// TIA Portal V21 export
FUNCTION_BLOCK "FB310"   // FB310, LAD
TITLE = FB310
{ S7_Optimized_Access := 'TRUE' }
AUTHOR : PRECISE
FAMILY : PRECISE
// RAW MATERIAL ADDITION 
// 0-MANUAL/1-SUCTION/2-LIQUID DRUM
// stored: AutoNumber false, MemoryReserve 100, SetENOAutomatically false
   VAR_INPUT
      Enable : Bool;
      Disable : Bool;
      Fault : Bool;
      SecPulse : Bool;
      AlwaysTrue : Bool;
      StartConfirmationPopupSel : Bool;   // StartConfirmationPopupSel: 0-NO/1-YES
      EndConfirmationPopupSel : Bool;   // EndConfirmationPopupSel: 0-NO/1-YES
      RMAddTypeSel : Int;   // RMAddTypeSel: 0-Manual/1-Suction/2-Liquid Drum
      RMTypeSel : Int := 1;   // RM Type Sel: Graules or Flakes -0/FinePowder-1
      WeightBasedSel : Bool;   // Weight Based Sel: 0-NO/1-YES
      AdditionMethodSel : Bool;   // Addition Method : 0-Add In Weight/1-Loss In Weight
      RMAddPopupSel : Bool;   // RM Add Popup Sel: 0-NO/1-YES
      SetRMNo : Int := 1;
      "SetVacuum/SetPressure" : Real := -300.0;   // SetVauum - For unit "mmHg" / SetPressure - For unit "bar"
      SetQuantity : Real := 10.0;   // Weight Based Sel: 1-YES
      SetSpeed : Real := 50.0;
      "ActualVacuum/ActualPressure" : Real;   // ActualVauum - For unit "mmHg" / ActualPressure - For unit "bar"
      ActualQuantity : Real;   // Collecting Vessel Weight
      ActualQuantityRMVessel : Real;   // Transffering Vessel Weight
      "VacuumTol/PressureTol" : Real := 10.0;   // VacuumTol - For unit "mmHg" / PressureTol - For unit "bar"
      DelaytoSettleMaterial : Int := 5;
      InflightQuantitySuction : Real;
      InflightQuantityLiqDrum : Real;
      DelaytoStartPump : Int := 3;
   END_VAR
   VAR_OUTPUT
      VacuumInValve : Bool;
      VacuumLineValves : Bool;
      SuctionInValve : Bool;
      VacuumPumpCmd : Bool;
      LineValves : Bool;
      PumpCmd : Bool;
      StartConfirmationPopup : Bool;   // For Start Confirmation Popup Selection: Yes
      EndConfirmationPopup : Bool;   // For End Confirmation Popup Selection: Yes
      DelaytoSettleMaterialPopup : Bool;   // "WAITING FOR MATERIAL TO SETTLE"
      RMAddPopup : Bool;   // For RMAddPopupSel: 1-YES
      RMAddPopupManual : Bool;   // For RMAddPopupSel: 1-YES
      ActualSpeed : Real;
      VisibleRM1 : Bool;
      VisibleRM2 : Bool;
      VisibleRM3 : Bool;
      VisibleRM4 : Bool;
      VisibleRM5 : Bool;
      VisibleRM6 : Bool;
      VisibleRM7 : Bool;
      VisibleRM8 : Bool;
      VisibleRM9 : Bool;
      VisibleRM10 : Bool;
      PrintTrigger : Bool;
      PrintWord : Int;
      PrintStatus : String[50];
   END_VAR
   VAR_IN_OUT
      Start : Bool;
      Stop : Bool;
      Reset : Bool;
      StartConfirmationAck : Bool;   // For Start Confirmation Popup Selection: Yes
      EndConfirmationAck : Bool;   // For End Confirmation Popup Selection: Yes
      SpareBtn1 : Bool;
      SpareBtn2 : Bool;
      Running : Bool;
      Selected : Bool;
      Paused : Bool;
      StartConfirmationPopupTemp : Bool;   // For Start Confirmation Popup Selection: Yes
      EndConfirmationPopupTemp : Bool;   // For End Confirmation Popup Selection: Yes
      RMAddPopupTemp : Bool;   // For RMAddPopupSel: 1-YES
      RMAddStarted : Bool;
      RMAddOver : Bool;
      ActualSetQuantityCalc : Real;   // For WeightBaseSel: 1-YES
      ActualSetQuantity : Real;   // For WeightBaseSel: 1-YES
      RMAddAck1 : Bool;   // For RMAddPopupSel: 1-YES
      RMAddAck2 : Bool;   // For RMAddPopupSel: 1-YES
      RMAddAck3 : Bool;   // For RMAddPopupSel: 1-YES
      RMAddAck4 : Bool;   // For RMAddPopupSel: 1-YES
      RMAddAck5 : Bool;   // For RMAddPopupSel: 1-YES
      RMAddAck6 : Bool;   // For RMAddPopupSel: 1-YES
      RMAddAck7 : Bool;   // For RMAddPopupSel: 1-YES
      RMAddAck8 : Bool;   // For RMAddPopupSel: 1-YES
      RMAddAck9 : Bool;   // For RMAddPopupSel: 1-YES
      RMAddAck10 : Bool;   // For RMAddPopupSel: 1-YES
   END_VAR
   VAR
      PrintTriggerTemp : Bool;
      RE1 : Bool;
      RE2 : Bool;
      RE3 : Bool;
      RE4 : Bool;
      RE5 : Bool;
      RE6 : Bool;
      RE7 : Bool;
      RE8 : Bool;
      RE9 : Bool;
      RE10 : Bool;
      RE11 : Bool;
      PrintTriggerResetTimer { S7_SetPoint := 'True'} : TON_TIME;
      BtnResetTimer { S7_SetPoint := 'True'} : TON_TIME;
   END_VAR
   VAR RETAIN
      NameRM1 : String[100];
   END_VAR
   VAR
      NameRM2 : String[100];
      NameRM3 : String[100];
      NameRM4 : String[100];
      NameRM5 : String[100];
      NameRM6 : String[100];
      NameRM7 : String[100];
      NameRM8 : String[100];
      NameRM9 : String[100];
      NameRM10 : String[100];
      Manual { S7_SetPoint := 'True'} : "FB307";
      Suction { S7_SetPoint := 'True'} : "FB308";
      LiqDrum { S7_SetPoint := 'True'} : "FB309";
   END_VAR
   VAR_TEMP
      STATUS1 : String[40];
      STATUS2 : String[40];
      STATUS3 : String[40];
      STATUS4 : String[40];
      STATUS5 : String[40];
      Blank : String[40];
   END_VAR
   VAR_TEMP   // added for the SCL form of the ladder/FBD networks
      _w1 : Bool;
      _w2 : Bool;
      _w3 : Bool;
      _w4 : Bool;
      _w5 : Bool;
      _w6 : Bool;
   END_VAR
BEGIN

REGION Network 1: Running
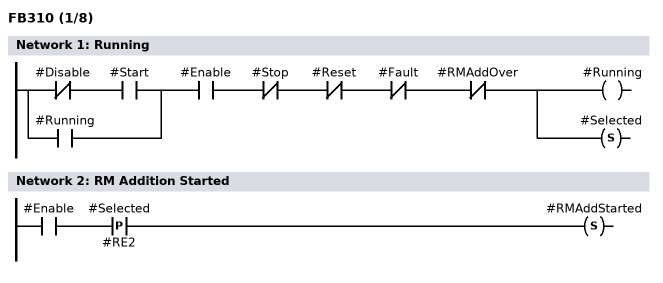
   RUNG wire#powerrail
      I_Contact( #Disable )
      Contact( #Start )
      wire#w1
      Contact( #Enable )
      I_Contact( #Stop )
      I_Contact( #Reset )
      I_Contact( #Fault )
      I_Contact( #RMAddOver )
      wire#w2
      Coil( #Running )
   END_RUNG
   RUNG wire#powerrail
      Contact( #Running )
   END_RUNG wire#w1
   RUNG wire#w2
      S_Coil( #Selected )
   END_RUNG
   // the same network as SCL:
   #Running := ((NOT #Disable AND #Start) OR #Running) AND #Enable AND NOT #Stop AND NOT #Reset AND NOT #Fault AND NOT #RMAddOver;
   IF #Running THEN #Selected := TRUE; END_IF;
END_REGION

REGION Network 2: RM Addition Started
   RUNG wire#powerrail
      Contact( #Enable )
      P_Contact(operand := #Selected, bit := #RE2)
      S_Coil( #RMAddStarted )
   END_RUNG
   // the same network as SCL:
   #_w1 := #Enable AND #Selected AND NOT #RE2;   // rising edge of #Selected
   #RE2 := #Selected;
   IF #_w1 THEN #RMAddStarted := TRUE; END_IF;
END_REGION

REGION Network 3: RM Addition Parameters
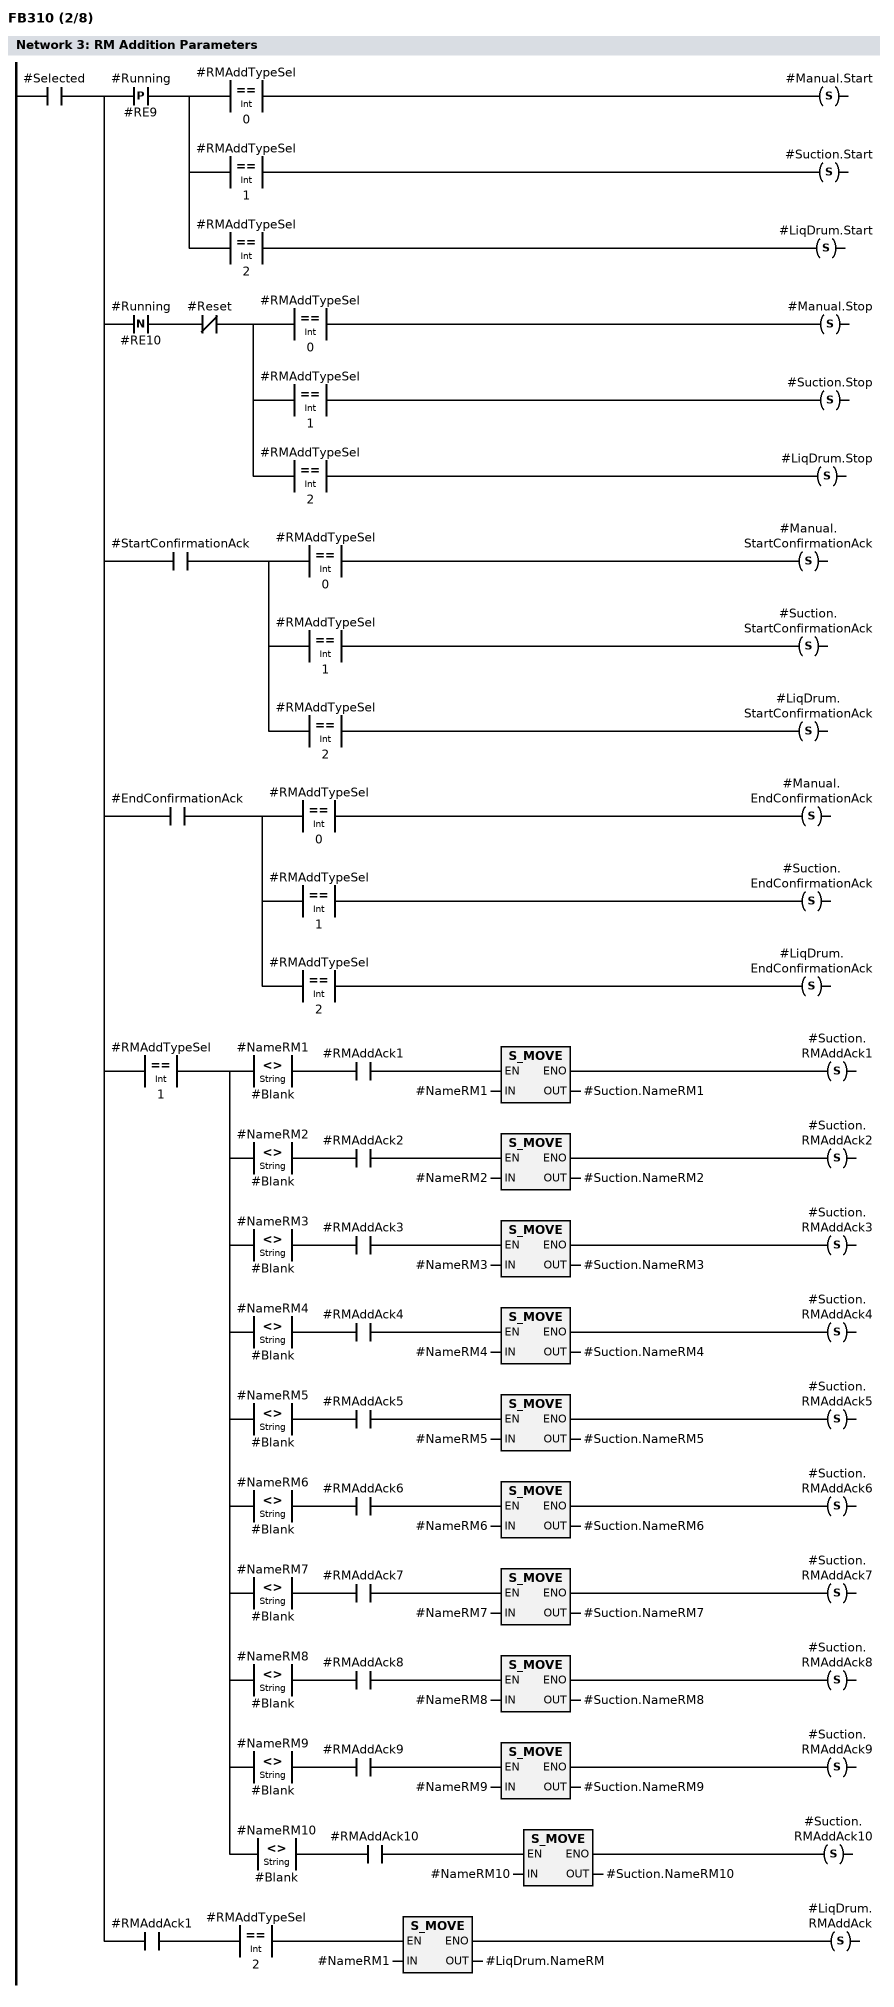
   RUNG wire#powerrail
      Contact( #Selected )
      wire#w1
      P_Contact(operand := #Running, bit := #RE9)
      wire#w2
      { S7_Templates := "SrcType := Int" } EQ_Contact(in1 := #RMAddTypeSel, in2 := 0)
      S_Coil( #Manual.Start )
   END_RUNG
   RUNG wire#w2
      { S7_Templates := "SrcType := Int" } EQ_Contact(in1 := #RMAddTypeSel, in2 := 1)
      S_Coil( #Suction.Start )
   END_RUNG
   RUNG wire#w2
      { S7_Templates := "SrcType := Int" } EQ_Contact(in1 := #RMAddTypeSel, in2 := 2)
      S_Coil( #LiqDrum.Start )
   END_RUNG
   RUNG wire#w1
      N_Contact(operand := #Running, bit := #RE10)
      I_Contact( #Reset )
      wire#w3
      { S7_Templates := "SrcType := Int" } EQ_Contact(in1 := #RMAddTypeSel, in2 := 0)
      S_Coil( #Manual.Stop )
   END_RUNG
   RUNG wire#w3
      { S7_Templates := "SrcType := Int" } EQ_Contact(in1 := #RMAddTypeSel, in2 := 1)
      S_Coil( #Suction.Stop )
   END_RUNG
   RUNG wire#w3
      { S7_Templates := "SrcType := Int" } EQ_Contact(in1 := #RMAddTypeSel, in2 := 2)
      S_Coil( #LiqDrum.Stop )
   END_RUNG
   RUNG wire#w1
      Contact( #StartConfirmationAck )
      wire#w4
      { S7_Templates := "SrcType := Int" } EQ_Contact(in1 := #RMAddTypeSel, in2 := 0)
      S_Coil( #Manual.StartConfirmationAck )
   END_RUNG
   RUNG wire#w4
      { S7_Templates := "SrcType := Int" } EQ_Contact(in1 := #RMAddTypeSel, in2 := 1)
      S_Coil( #Suction.StartConfirmationAck )
   END_RUNG
   RUNG wire#w4
      { S7_Templates := "SrcType := Int" } EQ_Contact(in1 := #RMAddTypeSel, in2 := 2)
      S_Coil( #LiqDrum.StartConfirmationAck )
   END_RUNG
   RUNG wire#w1
      Contact( #EndConfirmationAck )
      wire#w5
      { S7_Templates := "SrcType := Int" } EQ_Contact(in1 := #RMAddTypeSel, in2 := 0)
      S_Coil( #Manual.EndConfirmationAck )
   END_RUNG
   RUNG wire#w5
      { S7_Templates := "SrcType := Int" } EQ_Contact(in1 := #RMAddTypeSel, in2 := 1)
      S_Coil( #Suction.EndConfirmationAck )
   END_RUNG
   RUNG wire#w5
      { S7_Templates := "SrcType := Int" } EQ_Contact(in1 := #RMAddTypeSel, in2 := 2)
      S_Coil( #LiqDrum.EndConfirmationAck )
   END_RUNG
   RUNG wire#w1
      { S7_Templates := "SrcType := Int" } EQ_Contact(in1 := #RMAddTypeSel, in2 := 1)
      wire#w6
      { S7_Templates := "SrcType := String" } NE_Contact(in1 := #NameRM1, in2 := #Blank)
      Contact( #RMAddAck1 )
      S_Move(in := #NameRM1, out => #Suction.NameRM1)
      S_Coil( #Suction.RMAddAck1 )
   END_RUNG
   RUNG wire#w6
      { S7_Templates := "SrcType := String" } NE_Contact(in1 := #NameRM2, in2 := #Blank)
      Contact( #RMAddAck2 )
      S_Move(in := #NameRM2, out => #Suction.NameRM2)
      S_Coil( #Suction.RMAddAck2 )
   END_RUNG
   RUNG wire#w6
      { S7_Templates := "SrcType := String" } NE_Contact(in1 := #NameRM3, in2 := #Blank)
      Contact( #RMAddAck3 )
      S_Move(in := #NameRM3, out => #Suction.NameRM3)
      S_Coil( #Suction.RMAddAck3 )
   END_RUNG
   RUNG wire#w6
      { S7_Templates := "SrcType := String" } NE_Contact(in1 := #NameRM4, in2 := #Blank)
      Contact( #RMAddAck4 )
      S_Move(in := #NameRM4, out => #Suction.NameRM4)
      S_Coil( #Suction.RMAddAck4 )
   END_RUNG
   RUNG wire#w6
      { S7_Templates := "SrcType := String" } NE_Contact(in1 := #NameRM5, in2 := #Blank)
      Contact( #RMAddAck5 )
      S_Move(in := #NameRM5, out => #Suction.NameRM5)
      S_Coil( #Suction.RMAddAck5 )
   END_RUNG
   RUNG wire#w6
      { S7_Templates := "SrcType := String" } NE_Contact(in1 := #NameRM6, in2 := #Blank)
      Contact( #RMAddAck6 )
      S_Move(in := #NameRM6, out => #Suction.NameRM6)
      S_Coil( #Suction.RMAddAck6 )
   END_RUNG
   RUNG wire#w6
      { S7_Templates := "SrcType := String" } NE_Contact(in1 := #NameRM7, in2 := #Blank)
      Contact( #RMAddAck7 )
      S_Move(in := #NameRM7, out => #Suction.NameRM7)
      S_Coil( #Suction.RMAddAck7 )
   END_RUNG
   RUNG wire#w6
      { S7_Templates := "SrcType := String" } NE_Contact(in1 := #NameRM8, in2 := #Blank)
      Contact( #RMAddAck8 )
      S_Move(in := #NameRM8, out => #Suction.NameRM8)
      S_Coil( #Suction.RMAddAck8 )
   END_RUNG
   RUNG wire#w6
      { S7_Templates := "SrcType := String" } NE_Contact(in1 := #NameRM9, in2 := #Blank)
      Contact( #RMAddAck9 )
      S_Move(in := #NameRM9, out => #Suction.NameRM9)
      S_Coil( #Suction.RMAddAck9 )
   END_RUNG
   RUNG wire#w6
      { S7_Templates := "SrcType := String" } NE_Contact(in1 := #NameRM10, in2 := #Blank)
      Contact( #RMAddAck10 )
      S_Move(in := #NameRM10, out => #Suction.NameRM10)
      S_Coil( #Suction.RMAddAck10 )
   END_RUNG
   RUNG wire#w1
      Contact( #RMAddAck1 )
      { S7_Templates := "SrcType := Int" } EQ_Contact(in1 := #RMAddTypeSel, in2 := 2)
      S_Move(in := #NameRM1, out => #LiqDrum.NameRM)
      S_Coil( #LiqDrum.RMAddAck )
   END_RUNG
   // the same network as SCL:
   #_w1 := #Selected AND #Running AND NOT #RE9;   // rising edge of #Running
   #RE9 := #Running;
   IF #_w1 AND (#RMAddTypeSel = 0) THEN #Manual.Start := TRUE; END_IF;
   IF #_w1 AND (#RMAddTypeSel = 1) THEN #Suction.Start := TRUE; END_IF;
   IF #_w1 AND (#RMAddTypeSel = 2) THEN #LiqDrum.Start := TRUE; END_IF;
   #_w2 := #Selected AND NOT #Running AND #RE10;   // falling edge of #Running
   #RE10 := #Running;
   #_w3 := #_w2 AND NOT #Reset;
   IF #_w3 AND (#RMAddTypeSel = 0) THEN #Manual.Stop := TRUE; END_IF;
   IF #_w3 AND (#RMAddTypeSel = 1) THEN #Suction.Stop := TRUE; END_IF;
   IF #_w3 AND (#RMAddTypeSel = 2) THEN #LiqDrum.Stop := TRUE; END_IF;
   #_w4 := #Selected AND #StartConfirmationAck;
   IF #_w4 AND (#RMAddTypeSel = 0) THEN #Manual.StartConfirmationAck := TRUE; END_IF;
   IF #_w4 AND (#RMAddTypeSel = 1) THEN #Suction.StartConfirmationAck := TRUE; END_IF;
   IF #_w4 AND (#RMAddTypeSel = 2) THEN #LiqDrum.StartConfirmationAck := TRUE; END_IF;
   #_w5 := #Selected AND #EndConfirmationAck;
   IF #_w5 AND (#RMAddTypeSel = 0) THEN #Manual.EndConfirmationAck := TRUE; END_IF;
   IF #_w5 AND (#RMAddTypeSel = 1) THEN #Suction.EndConfirmationAck := TRUE; END_IF;
   IF #_w5 AND (#RMAddTypeSel = 2) THEN #LiqDrum.EndConfirmationAck := TRUE; END_IF;
   #_w6 := #Selected AND (#RMAddTypeSel = 1);
   IF #_w6 AND (#NameRM1 <> #Blank) AND #RMAddAck1 THEN
       #Suction.NameRM1 := #NameRM1;
       #Suction.RMAddAck1 := TRUE;
   END_IF;
   IF #_w6 AND (#NameRM2 <> #Blank) AND #RMAddAck2 THEN
       #Suction.NameRM2 := #NameRM2;
       #Suction.RMAddAck2 := TRUE;
   END_IF;
   IF #_w6 AND (#NameRM3 <> #Blank) AND #RMAddAck3 THEN
       #Suction.NameRM3 := #NameRM3;
       #Suction.RMAddAck3 := TRUE;
   END_IF;
   IF #_w6 AND (#NameRM4 <> #Blank) AND #RMAddAck4 THEN
       #Suction.NameRM4 := #NameRM4;
       #Suction.RMAddAck4 := TRUE;
   END_IF;
   IF #_w6 AND (#NameRM5 <> #Blank) AND #RMAddAck5 THEN
       #Suction.NameRM5 := #NameRM5;
       #Suction.RMAddAck5 := TRUE;
   END_IF;
   IF #_w6 AND (#NameRM6 <> #Blank) AND #RMAddAck6 THEN
       #Suction.NameRM6 := #NameRM6;
       #Suction.RMAddAck6 := TRUE;
   END_IF;
   IF #_w6 AND (#NameRM7 <> #Blank) AND #RMAddAck7 THEN
       #Suction.NameRM7 := #NameRM7;
       #Suction.RMAddAck7 := TRUE;
   END_IF;
   IF #_w6 AND (#NameRM8 <> #Blank) AND #RMAddAck8 THEN
       #Suction.NameRM8 := #NameRM8;
       #Suction.RMAddAck8 := TRUE;
   END_IF;
   IF #_w6 AND (#NameRM9 <> #Blank) AND #RMAddAck9 THEN
       #Suction.NameRM9 := #NameRM9;
       #Suction.RMAddAck9 := TRUE;
   END_IF;
   IF #_w6 AND (#NameRM10 <> #Blank) AND #RMAddAck10 THEN
       #Suction.NameRM10 := #NameRM10;
       #Suction.RMAddAck10 := TRUE;
   END_IF;
   IF #Selected AND #RMAddAck1 AND (#RMAddTypeSel = 2) THEN
       #LiqDrum.NameRM := #NameRM1;
       #LiqDrum.RMAddAck := TRUE;
   END_IF;
END_REGION

REGION Network 4: RM Addition Manual
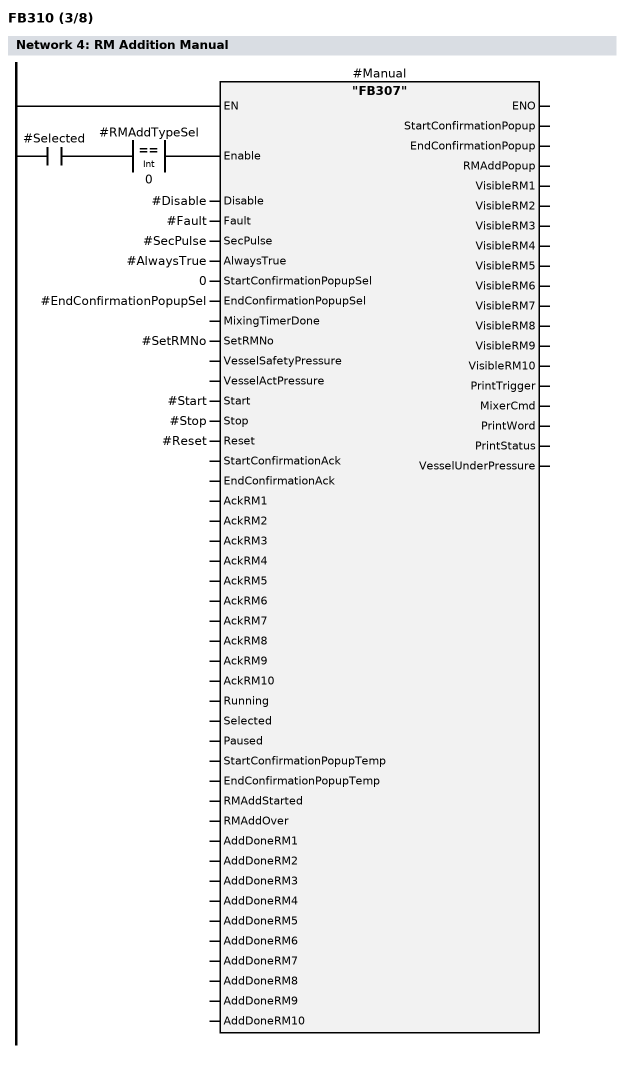
   RUNG wire#powerrail
      #Manual(Enable := wire#w1, Disable := #Disable, Fault := #Fault, SecPulse := #SecPulse, AlwaysTrue := #AlwaysTrue, StartConfirmationPopupSel := 0, EndConfirmationPopupSel := #EndConfirmationPopupSel, MixingTimerDone :=, SetRMNo := #SetRMNo, VesselSafetyPressure :=, VesselActPressure :=, Start := #Start, Stop := #Stop, Reset := #Reset, StartConfirmationAck :=, EndConfirmationAck :=, AckRM1 :=, AckRM2 :=, AckRM3 :=, AckRM4 :=, AckRM5 :=, AckRM6 :=, AckRM7 :=, AckRM8 :=, AckRM9 :=, AckRM10 :=, Running :=, Selected :=, Paused :=, StartConfirmationPopupTemp :=, EndConfirmationPopupTemp :=, RMAddStarted :=, RMAddOver :=, AddDoneRM1 :=, AddDoneRM2 :=, AddDoneRM3 :=, AddDoneRM4 :=, AddDoneRM5 :=, AddDoneRM6 :=, AddDoneRM7 :=, AddDoneRM8 :=, AddDoneRM9 :=, AddDoneRM10 :=, StartConfirmationPopup =>, EndConfirmationPopup =>, RMAddPopup =>, VisibleRM1 =>, VisibleRM2 =>, VisibleRM3 =>, VisibleRM4 =>, VisibleRM5 =>, VisibleRM6 =>, VisibleRM7 =>, VisibleRM8 =>, VisibleRM9 =>, VisibleRM10 =>, PrintTrigger =>, MixerCmd =>, PrintWord =>, PrintStatus =>, VesselUnderPressure =>)
   END_RUNG
   RUNG wire#powerrail
      Contact( #Selected )
      { S7_Templates := "SrcType := Int" } EQ_Contact(in1 := #RMAddTypeSel, in2 := 0)
   END_RUNG wire#w1
   // the same network as SCL:
   #Manual(Enable := #Selected AND (#RMAddTypeSel = 0),   // "FB307"
           Disable := #Disable,
           Fault := #Fault,
           SecPulse := #SecPulse,
           AlwaysTrue := #AlwaysTrue,
           StartConfirmationPopupSel := 0,
           EndConfirmationPopupSel := #EndConfirmationPopupSel,
           SetRMNo := #SetRMNo,
           Start := #Start,
           Stop := #Stop,
           Reset := #Reset);
END_REGION

REGION Network 5: RM Addition Suction
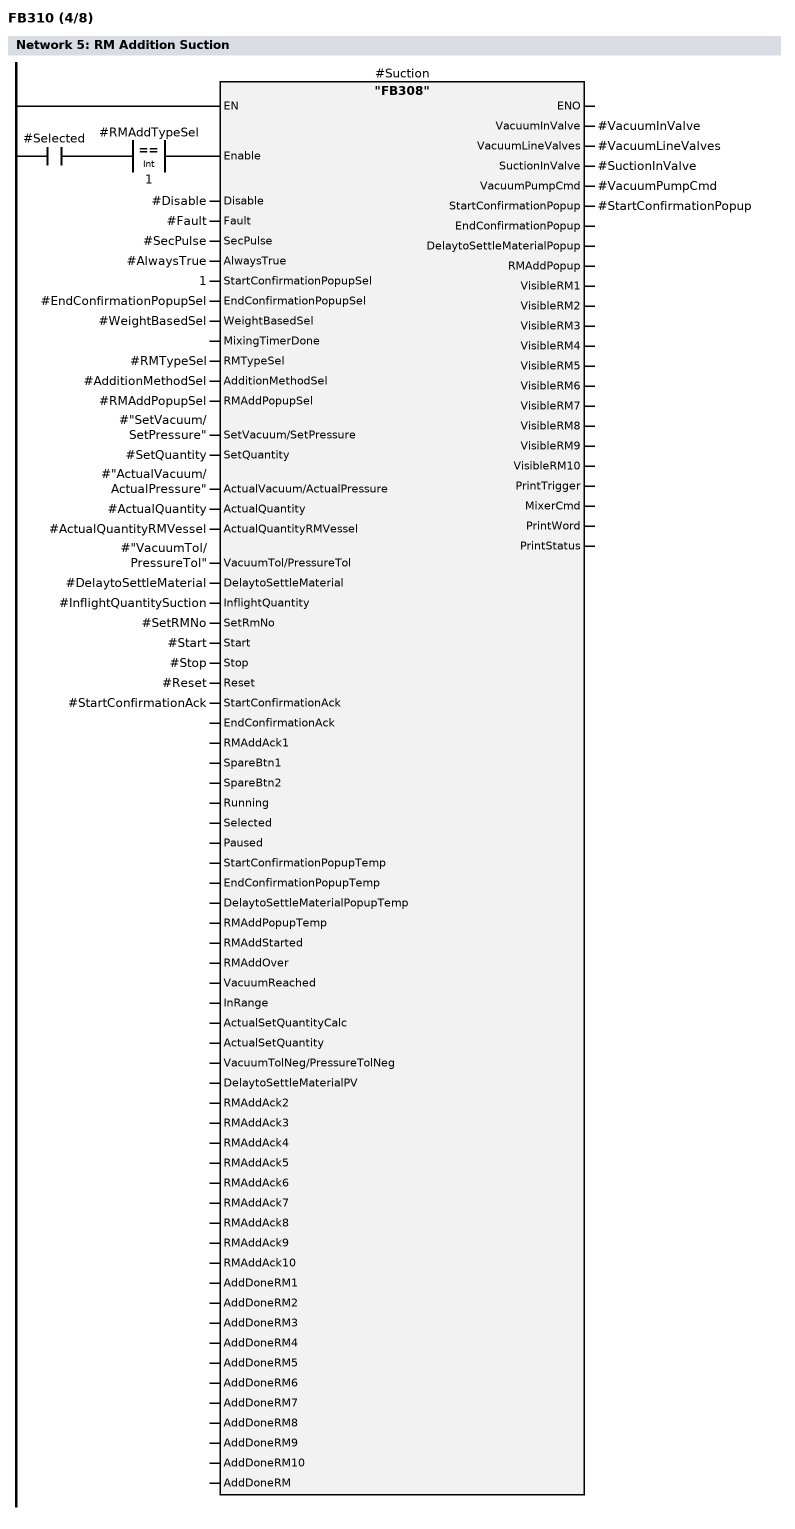
   RUNG wire#powerrail
      #Suction(Enable := wire#w1, Disable := #Disable, Fault := #Fault, SecPulse := #SecPulse, AlwaysTrue := #AlwaysTrue, StartConfirmationPopupSel := 1, EndConfirmationPopupSel := #EndConfirmationPopupSel, WeightBasedSel := #WeightBasedSel, MixingTimerDone :=, RMTypeSel := #RMTypeSel, AdditionMethodSel := #AdditionMethodSel, RMAddPopupSel := #RMAddPopupSel, "SetVacuum/SetPressure" := #"SetVacuum/SetPressure", SetQuantity := #SetQuantity, "ActualVacuum/ActualPressure" := #"ActualVacuum/ActualPressure", ActualQuantity := #ActualQuantity, ActualQuantityRMVessel := #ActualQuantityRMVessel, "VacuumTol/PressureTol" := #"VacuumTol/PressureTol", DelaytoSettleMaterial := #DelaytoSettleMaterial, InflightQuantity := #InflightQuantitySuction, SetRmNo := #SetRMNo, Start := #Start, Stop := #Stop, Reset := #Reset, StartConfirmationAck := #StartConfirmationAck, EndConfirmationAck :=, RMAddAck1 :=, SpareBtn1 :=, SpareBtn2 :=, Running :=, Selected :=, Paused :=, StartConfirmationPopupTemp :=, EndConfirmationPopupTemp :=, DelaytoSettleMaterialPopupTemp :=, RMAddPopupTemp :=, RMAddStarted :=, RMAddOver :=, VacuumReached :=, InRange :=, ActualSetQuantityCalc :=, ActualSetQuantity :=, "VacuumTolNeg/PressureTolNeg" :=, DelaytoSettleMaterialPV :=, RMAddAck2 :=, RMAddAck3 :=, RMAddAck4 :=, RMAddAck5 :=, RMAddAck6 :=, RMAddAck7 :=, RMAddAck8 :=, RMAddAck9 :=, RMAddAck10 :=, AddDoneRM1 :=, AddDoneRM2 :=, AddDoneRM3 :=, AddDoneRM4 :=, AddDoneRM5 :=, AddDoneRM6 :=, AddDoneRM7 :=, AddDoneRM8 :=, AddDoneRM9 :=, AddDoneRM10 :=, AddDoneRM :=, VacuumInValve => #VacuumInValve, VacuumLineValves => #VacuumLineValves, SuctionInValve => #SuctionInValve, VacuumPumpCmd => #VacuumPumpCmd, StartConfirmationPopup => #StartConfirmationPopup, EndConfirmationPopup =>, DelaytoSettleMaterialPopup =>, RMAddPopup =>, VisibleRM1 =>, VisibleRM2 =>, VisibleRM3 =>, VisibleRM4 =>, VisibleRM5 =>, VisibleRM6 =>, VisibleRM7 =>, VisibleRM8 =>, VisibleRM9 =>, VisibleRM10 =>, PrintTrigger =>, MixerCmd =>, PrintWord =>, PrintStatus =>)
   END_RUNG
   RUNG wire#powerrail
      Contact( #Selected )
      { S7_Templates := "SrcType := Int" } EQ_Contact(in1 := #RMAddTypeSel, in2 := 1)
   END_RUNG wire#w1
   // the same network as SCL:
   #Suction(Enable := #Selected AND (#RMAddTypeSel = 1),   // "FB308"
            Disable := #Disable,
            Fault := #Fault,
            SecPulse := #SecPulse,
            AlwaysTrue := #AlwaysTrue,
            StartConfirmationPopupSel := 1,
            EndConfirmationPopupSel := #EndConfirmationPopupSel,
            WeightBasedSel := #WeightBasedSel,
            RMTypeSel := #RMTypeSel,
            AdditionMethodSel := #AdditionMethodSel,
            RMAddPopupSel := #RMAddPopupSel,
            "SetVacuum/SetPressure" := #"SetVacuum/SetPressure",
            SetQuantity := #SetQuantity,
            "ActualVacuum/ActualPressure" := #"ActualVacuum/ActualPressure",
            ActualQuantity := #ActualQuantity,
            ActualQuantityRMVessel := #ActualQuantityRMVessel,
            "VacuumTol/PressureTol" := #"VacuumTol/PressureTol",
            DelaytoSettleMaterial := #DelaytoSettleMaterial,
            InflightQuantity := #InflightQuantitySuction,
            SetRmNo := #SetRMNo,
            Start := #Start,
            Stop := #Stop,
            Reset := #Reset,
            StartConfirmationAck := #StartConfirmationAck,
            VacuumInValve => #VacuumInValve,
            VacuumLineValves => #VacuumLineValves,
            SuctionInValve => #SuctionInValve,
            VacuumPumpCmd => #VacuumPumpCmd,
            StartConfirmationPopup => #StartConfirmationPopup);
END_REGION

REGION Network 6: RM Addition Liquid Drum
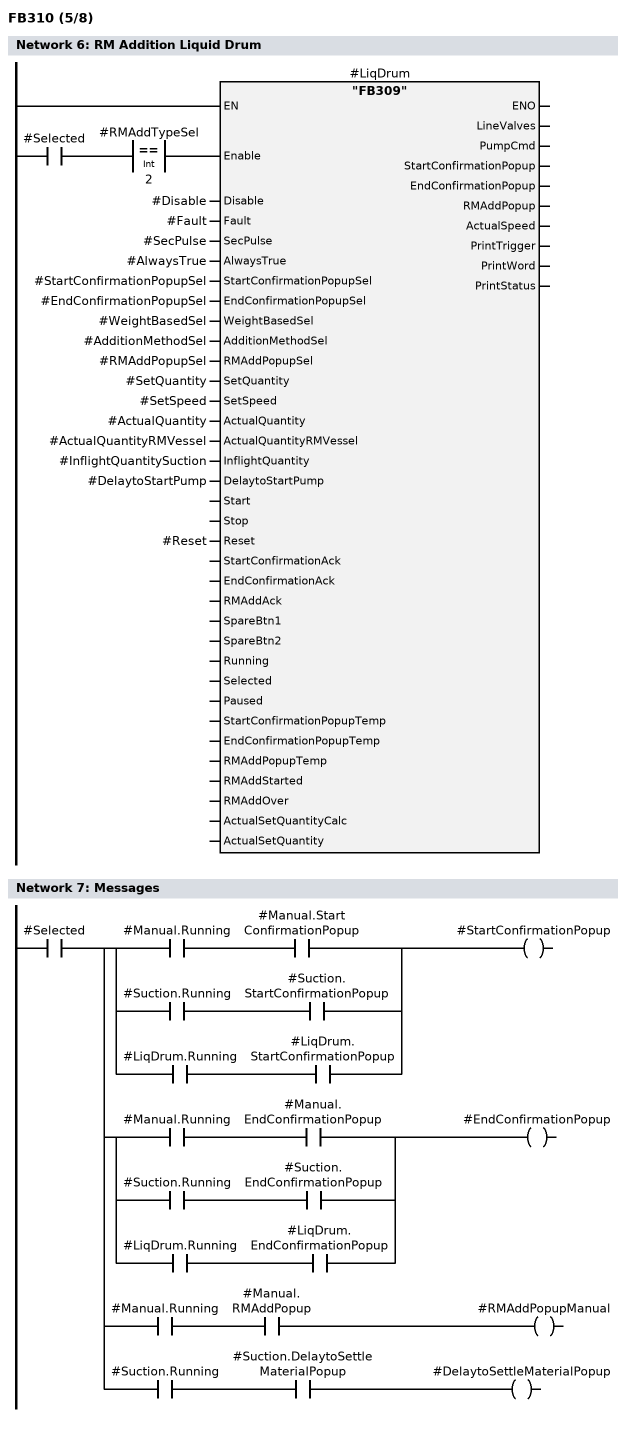
   RUNG wire#powerrail
      #LiqDrum(Enable := wire#w1, Disable := #Disable, Fault := #Fault, SecPulse := #SecPulse, AlwaysTrue := #AlwaysTrue, StartConfirmationPopupSel := #StartConfirmationPopupSel, EndConfirmationPopupSel := #EndConfirmationPopupSel, WeightBasedSel := #WeightBasedSel, AdditionMethodSel := #AdditionMethodSel, RMAddPopupSel := #RMAddPopupSel, SetQuantity := #SetQuantity, SetSpeed := #SetSpeed, ActualQuantity := #ActualQuantity, ActualQuantityRMVessel := #ActualQuantityRMVessel, InflightQuantity := #InflightQuantitySuction, DelaytoStartPump := #DelaytoStartPump, Start :=, Stop :=, Reset := #Reset, StartConfirmationAck :=, EndConfirmationAck :=, RMAddAck :=, SpareBtn1 :=, SpareBtn2 :=, Running :=, Selected :=, Paused :=, StartConfirmationPopupTemp :=, EndConfirmationPopupTemp :=, RMAddPopupTemp :=, RMAddStarted :=, RMAddOver :=, ActualSetQuantityCalc :=, ActualSetQuantity :=, LineValves =>, PumpCmd =>, StartConfirmationPopup =>, EndConfirmationPopup =>, RMAddPopup =>, ActualSpeed =>, PrintTrigger =>, PrintWord =>, PrintStatus =>)
   END_RUNG
   RUNG wire#powerrail
      Contact( #Selected )
      { S7_Templates := "SrcType := Int" } EQ_Contact(in1 := #RMAddTypeSel, in2 := 2)
   END_RUNG wire#w1
   // the same network as SCL:
   #LiqDrum(Enable := #Selected AND (#RMAddTypeSel = 2),   // "FB309"
            Disable := #Disable,
            Fault := #Fault,
            SecPulse := #SecPulse,
            AlwaysTrue := #AlwaysTrue,
            StartConfirmationPopupSel := #StartConfirmationPopupSel,
            EndConfirmationPopupSel := #EndConfirmationPopupSel,
            WeightBasedSel := #WeightBasedSel,
            AdditionMethodSel := #AdditionMethodSel,
            RMAddPopupSel := #RMAddPopupSel,
            SetQuantity := #SetQuantity,
            SetSpeed := #SetSpeed,
            ActualQuantity := #ActualQuantity,
            ActualQuantityRMVessel := #ActualQuantityRMVessel,
            InflightQuantity := #InflightQuantitySuction,
            DelaytoStartPump := #DelaytoStartPump,
            Reset := #Reset);
END_REGION

REGION Network 7: Messages
   RUNG wire#powerrail
      Contact( #Selected )
      wire#w1
      Contact( #Manual.Running )
      Contact( #Manual.StartConfirmationPopup )
      wire#w2
      Coil( #StartConfirmationPopup )
   END_RUNG
   RUNG wire#w1
      Contact( #Suction.Running )
      Contact( #Suction.StartConfirmationPopup )
   END_RUNG wire#w2
   RUNG wire#w1
      Contact( #LiqDrum.Running )
      Contact( #LiqDrum.StartConfirmationPopup )
   END_RUNG wire#w2
   RUNG wire#w1
      Contact( #Manual.Running )
      Contact( #Manual.EndConfirmationPopup )
      wire#w3
      Coil( #EndConfirmationPopup )
   END_RUNG
   RUNG wire#w1
      Contact( #Suction.Running )
      Contact( #Suction.EndConfirmationPopup )
   END_RUNG wire#w3
   RUNG wire#w1
      Contact( #LiqDrum.Running )
      Contact( #LiqDrum.EndConfirmationPopup )
   END_RUNG wire#w3
   RUNG wire#w1
      Contact( #Manual.Running )
      Contact( #Manual.RMAddPopup )
      Coil( #RMAddPopupManual )
   END_RUNG
   RUNG wire#w1
      Contact( #Suction.Running )
      Contact( #Suction.DelaytoSettleMaterialPopup )
      Coil( #DelaytoSettleMaterialPopup )
   END_RUNG
   // the same network as SCL:
   #StartConfirmationPopup := #Selected AND ((#Manual.Running AND #Manual.StartConfirmationPopup) OR (#Suction.Running AND #Suction.StartConfirmationPopup) OR (#LiqDrum.Running AND #LiqDrum.StartConfirmationPopup));
   #EndConfirmationPopup := #Selected AND ((#Manual.Running AND #Manual.EndConfirmationPopup) OR (#Suction.Running AND #Suction.EndConfirmationPopup) OR (#LiqDrum.Running AND #LiqDrum.EndConfirmationPopup));
   #RMAddPopupManual := #Selected AND #Manual.Running AND #Manual.RMAddPopup;
   #DelaytoSettleMaterialPopup := #Selected AND #Suction.Running AND #Suction.DelaytoSettleMaterialPopup;
END_REGION

REGION Network 8: Output
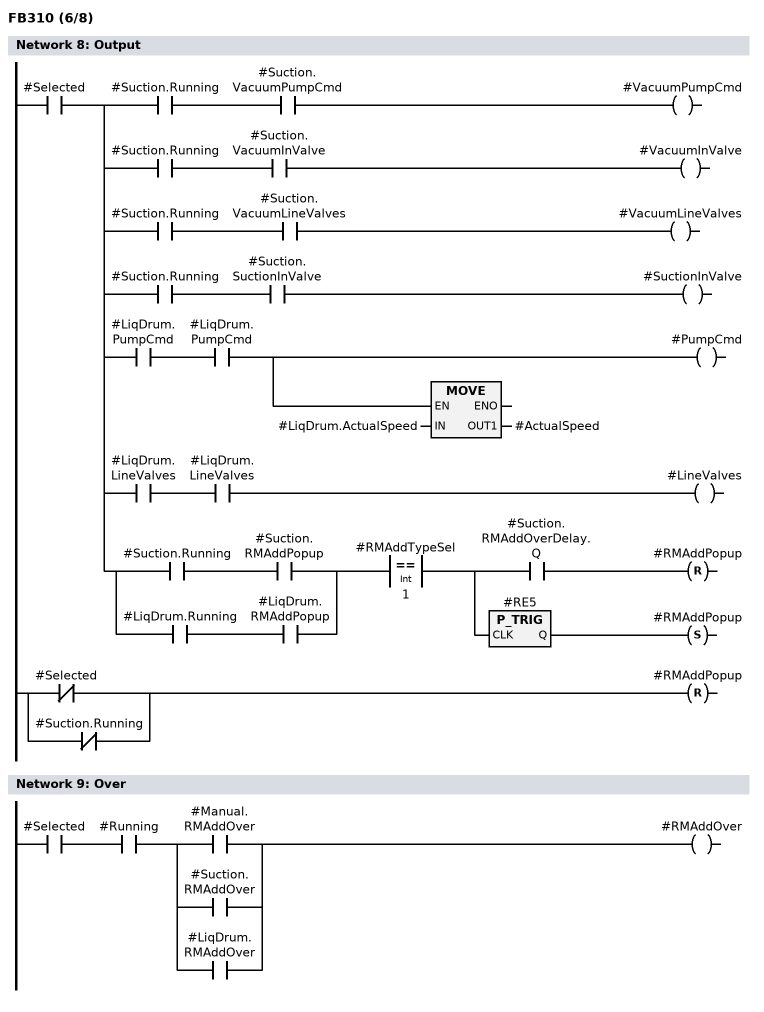
   RUNG wire#powerrail
      Contact( #Selected )
      wire#w1
      Contact( #Suction.Running )
      Contact( #Suction.VacuumPumpCmd )
      Coil( #VacuumPumpCmd )
   END_RUNG
   RUNG wire#w1
      Contact( #Suction.Running )
      Contact( #Suction.VacuumInValve )
      Coil( #VacuumInValve )
   END_RUNG
   RUNG wire#w1
      Contact( #Suction.Running )
      Contact( #Suction.VacuumLineValves )
      Coil( #VacuumLineValves )
   END_RUNG
   RUNG wire#w1
      Contact( #Suction.Running )
      Contact( #Suction.SuctionInValve )
      Coil( #SuctionInValve )
   END_RUNG
   RUNG wire#w1
      Contact( #LiqDrum.PumpCmd )
      Contact( #LiqDrum.PumpCmd )
      wire#w2
      Coil( #PumpCmd )
   END_RUNG
   RUNG wire#w2
      Move(in := #LiqDrum.ActualSpeed, out1 => #ActualSpeed)
   END_RUNG
   RUNG wire#w1
      Contact( #LiqDrum.LineValves )
      Contact( #LiqDrum.LineValves )
      Coil( #LineValves )
   END_RUNG
   RUNG wire#w1
      Contact( #Suction.Running )
      Contact( #Suction.RMAddPopup )
      wire#w3
      { S7_Templates := "SrcType := Int" } EQ_Contact(in1 := #RMAddTypeSel, in2 := 1)
      wire#w4
      Contact( #Suction.RMAddOverDelay.Q )
      R_Coil( #RMAddPopup )
   END_RUNG
   RUNG wire#w1
      Contact( #LiqDrum.Running )
      Contact( #LiqDrum.RMAddPopup )
   END_RUNG wire#w3
   RUNG wire#w4
      P_Trig( #RE5 )
      S_Coil( #RMAddPopup )
   END_RUNG
   RUNG wire#powerrail
      I_Contact( #Selected )
      wire#w5
      R_Coil( #RMAddPopup )
   END_RUNG
   RUNG wire#powerrail
      I_Contact( #Suction.Running )
   END_RUNG wire#w5
   // the same network as SCL:
   #VacuumPumpCmd := #Selected AND #Suction.Running AND #Suction.VacuumPumpCmd;
   #VacuumInValve := #Selected AND #Suction.Running AND #Suction.VacuumInValve;
   #VacuumLineValves := #Selected AND #Suction.Running AND #Suction.VacuumLineValves;
   #SuctionInValve := #Selected AND #Suction.Running AND #Suction.SuctionInValve;
   #PumpCmd := #Selected AND #LiqDrum.PumpCmd AND #LiqDrum.PumpCmd;
   IF #PumpCmd THEN #ActualSpeed := #LiqDrum.ActualSpeed; END_IF;
   #LineValves := #Selected AND #LiqDrum.LineValves AND #LiqDrum.LineValves;
   #_w1 := #Selected AND ((#Suction.Running AND #Suction.RMAddPopup) OR (#LiqDrum.Running AND #LiqDrum.RMAddPopup)) AND (#RMAddTypeSel = 1);
   IF #_w1 AND #Suction.RMAddOverDelay.Q THEN #RMAddPopup := FALSE; END_IF;
   #_w2 := #_w1 AND NOT #RE5;   // rising edge
   #RE5 := #_w1;
   IF #_w2 THEN #RMAddPopup := TRUE; END_IF;
   IF NOT #Selected OR NOT #Suction.Running THEN #RMAddPopup := FALSE; END_IF;
END_REGION

REGION Network 9: Over
   RUNG wire#powerrail
      Contact( #Selected )
      Contact( #Running )
      wire#w1
      Contact( #Manual.RMAddOver )
      wire#w2
      Coil( #RMAddOver )
   END_RUNG
   RUNG wire#w1
      Contact( #Suction.RMAddOver )
   END_RUNG wire#w2
   RUNG wire#w1
      Contact( #LiqDrum.RMAddOver )
   END_RUNG wire#w2
   // the same network as SCL:
   #RMAddOver := #Selected AND #Running AND (#Manual.RMAddOver OR #Suction.RMAddOver OR #LiqDrum.RMAddOver);
END_REGION

REGION Network 10: Print Status
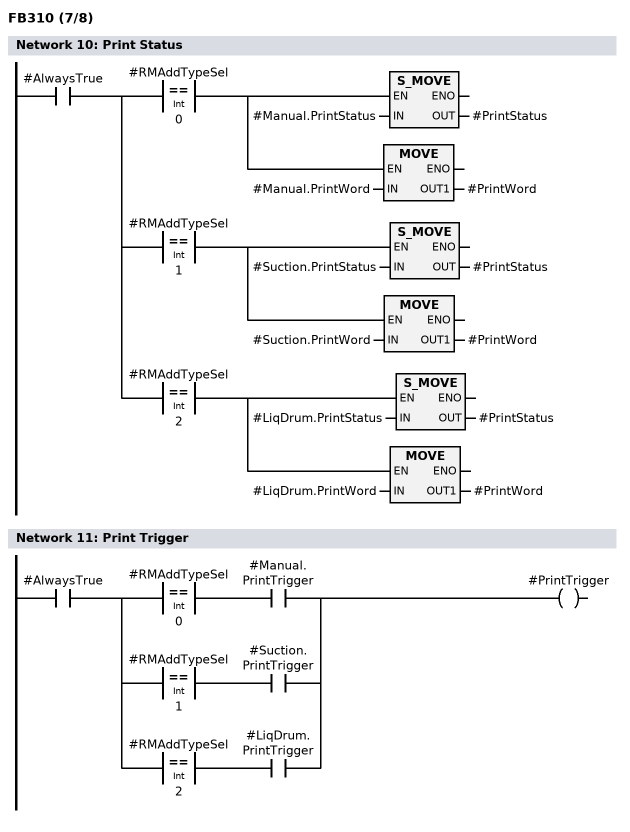
   RUNG wire#powerrail
      Contact( #AlwaysTrue )
      wire#w1
      { S7_Templates := "SrcType := Int" } EQ_Contact(in1 := #RMAddTypeSel, in2 := 0)
      wire#w2
      S_Move(in := #Manual.PrintStatus, out => #PrintStatus)
   END_RUNG
   RUNG wire#w2
      Move(in := #Manual.PrintWord, out1 => #PrintWord)
   END_RUNG
   RUNG wire#w1
      { S7_Templates := "SrcType := Int" } EQ_Contact(in1 := #RMAddTypeSel, in2 := 1)
      wire#w3
      S_Move(in := #Suction.PrintStatus, out => #PrintStatus)
   END_RUNG
   RUNG wire#w3
      Move(in := #Suction.PrintWord, out1 => #PrintWord)
   END_RUNG
   RUNG wire#w1
      { S7_Templates := "SrcType := Int" } EQ_Contact(in1 := #RMAddTypeSel, in2 := 2)
      wire#w4
      S_Move(in := #LiqDrum.PrintStatus, out => #PrintStatus)
   END_RUNG
   RUNG wire#w4
      Move(in := #LiqDrum.PrintWord, out1 => #PrintWord)
   END_RUNG
   // the same network as SCL:
   IF #AlwaysTrue AND (#RMAddTypeSel = 0) THEN
       #PrintStatus := #Manual.PrintStatus;
       #PrintWord := #Manual.PrintWord;
   END_IF;
   IF #AlwaysTrue AND (#RMAddTypeSel = 1) THEN
       #PrintStatus := #Suction.PrintStatus;
       #PrintWord := #Suction.PrintWord;
   END_IF;
   IF #AlwaysTrue AND (#RMAddTypeSel = 2) THEN
       #PrintStatus := #LiqDrum.PrintStatus;
       #PrintWord := #LiqDrum.PrintWord;
   END_IF;
END_REGION

REGION Network 11: Print Trigger
   RUNG wire#powerrail
      Contact( #AlwaysTrue )
      wire#w1
      { S7_Templates := "SrcType := Int" } EQ_Contact(in1 := #RMAddTypeSel, in2 := 0)
      Contact( #Manual.PrintTrigger )
      wire#w2
      Coil( #PrintTrigger )
   END_RUNG
   RUNG wire#w1
      { S7_Templates := "SrcType := Int" } EQ_Contact(in1 := #RMAddTypeSel, in2 := 1)
      Contact( #Suction.PrintTrigger )
   END_RUNG wire#w2
   RUNG wire#w1
      { S7_Templates := "SrcType := Int" } EQ_Contact(in1 := #RMAddTypeSel, in2 := 2)
      Contact( #LiqDrum.PrintTrigger )
   END_RUNG wire#w2
   // the same network as SCL:
   #PrintTrigger := #AlwaysTrue AND (((#RMAddTypeSel = 0) AND #Manual.PrintTrigger) OR ((#RMAddTypeSel = 1) AND #Suction.PrintTrigger) OR ((#RMAddTypeSel = 2) AND #LiqDrum.PrintTrigger));
END_REGION

REGION Network 12: Button Reset
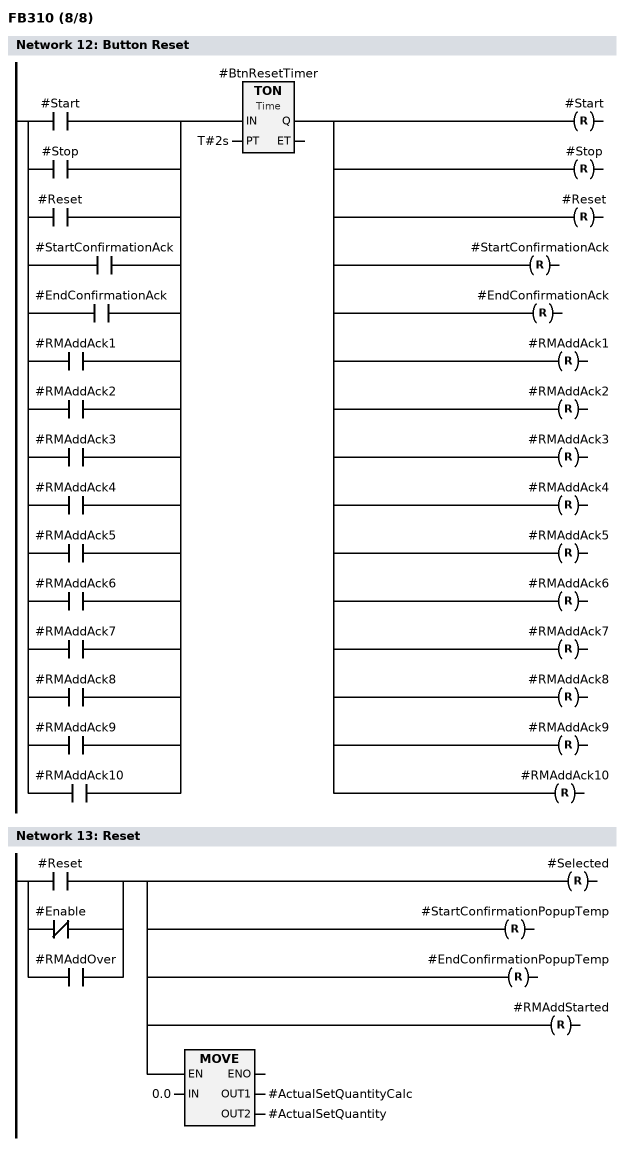
   RUNG wire#powerrail
      Contact( #Start )
      wire#w1
      { S7_Templates := "time_type := Time" } #BtnResetTimer.TON(pt := T#2s, et =>)
      wire#w2
      R_Coil( #Start )
   END_RUNG
   RUNG wire#powerrail
      Contact( #Stop )
   END_RUNG wire#w1
   RUNG wire#powerrail
      Contact( #Reset )
   END_RUNG wire#w1
   RUNG wire#powerrail
      Contact( #StartConfirmationAck )
   END_RUNG wire#w1
   RUNG wire#powerrail
      Contact( #EndConfirmationAck )
   END_RUNG wire#w1
   RUNG wire#powerrail
      Contact( #RMAddAck1 )
   END_RUNG wire#w1
   RUNG wire#powerrail
      Contact( #RMAddAck2 )
   END_RUNG wire#w1
   RUNG wire#powerrail
      Contact( #RMAddAck3 )
   END_RUNG wire#w1
   RUNG wire#powerrail
      Contact( #RMAddAck4 )
   END_RUNG wire#w1
   RUNG wire#powerrail
      Contact( #RMAddAck5 )
   END_RUNG wire#w1
   RUNG wire#powerrail
      Contact( #RMAddAck6 )
   END_RUNG wire#w1
   RUNG wire#powerrail
      Contact( #RMAddAck7 )
   END_RUNG wire#w1
   RUNG wire#powerrail
      Contact( #RMAddAck8 )
   END_RUNG wire#w1
   RUNG wire#powerrail
      Contact( #RMAddAck9 )
   END_RUNG wire#w1
   RUNG wire#powerrail
      Contact( #RMAddAck10 )
   END_RUNG wire#w1
   RUNG wire#w2
      R_Coil( #Stop )
   END_RUNG
   RUNG wire#w2
      R_Coil( #Reset )
   END_RUNG
   RUNG wire#w2
      R_Coil( #StartConfirmationAck )
   END_RUNG
   RUNG wire#w2
      R_Coil( #EndConfirmationAck )
   END_RUNG
   RUNG wire#w2
      R_Coil( #RMAddAck1 )
   END_RUNG
   RUNG wire#w2
      R_Coil( #RMAddAck2 )
   END_RUNG
   RUNG wire#w2
      R_Coil( #RMAddAck3 )
   END_RUNG
   RUNG wire#w2
      R_Coil( #RMAddAck4 )
   END_RUNG
   RUNG wire#w2
      R_Coil( #RMAddAck5 )
   END_RUNG
   RUNG wire#w2
      R_Coil( #RMAddAck6 )
   END_RUNG
   RUNG wire#w2
      R_Coil( #RMAddAck7 )
   END_RUNG
   RUNG wire#w2
      R_Coil( #RMAddAck8 )
   END_RUNG
   RUNG wire#w2
      R_Coil( #RMAddAck9 )
   END_RUNG
   RUNG wire#w2
      R_Coil( #RMAddAck10 )
   END_RUNG
   // the same network as SCL:
   #BtnResetTimer(IN := #Start OR #Stop OR #Reset OR #StartConfirmationAck OR #EndConfirmationAck OR #RMAddAck1 OR #RMAddAck2 OR #RMAddAck3 OR #RMAddAck4 OR #RMAddAck5 OR #RMAddAck6 OR #RMAddAck7 OR #RMAddAck8 OR #RMAddAck9 OR #RMAddAck10,   // TON
                  PT := T#2s);
   IF #BtnResetTimer.Q THEN
       #Start := FALSE;
       #Stop := FALSE;
       #Reset := FALSE;
       #StartConfirmationAck := FALSE;
       #EndConfirmationAck := FALSE;
       #RMAddAck1 := FALSE;
       #RMAddAck2 := FALSE;
       #RMAddAck3 := FALSE;
       #RMAddAck4 := FALSE;
       #RMAddAck5 := FALSE;
       #RMAddAck6 := FALSE;
       #RMAddAck7 := FALSE;
       #RMAddAck8 := FALSE;
       #RMAddAck9 := FALSE;
       #RMAddAck10 := FALSE;
   END_IF;
END_REGION

REGION Network 13: Reset
   RUNG wire#powerrail
      Contact( #Reset )
      wire#w1
      R_Coil( #Selected )
   END_RUNG
   RUNG wire#powerrail
      I_Contact( #Enable )
   END_RUNG wire#w1
   RUNG wire#powerrail
      Contact( #RMAddOver )
   END_RUNG wire#w1
   RUNG wire#w1
      R_Coil( #StartConfirmationPopupTemp )
   END_RUNG
   RUNG wire#w1
      R_Coil( #EndConfirmationPopupTemp )
   END_RUNG
   RUNG wire#w1
      R_Coil( #RMAddStarted )
   END_RUNG
   RUNG wire#w1
      Move(in := 0.0, out1 => #ActualSetQuantityCalc, out2 => #ActualSetQuantity)
   END_RUNG
   // the same network as SCL:
   IF #Reset OR NOT #Enable OR #RMAddOver THEN
       #Selected := FALSE;
       #StartConfirmationPopupTemp := FALSE;
       #EndConfirmationPopupTemp := FALSE;
       #RMAddStarted := FALSE;
       #ActualSetQuantityCalc := 0.0;
       #ActualSetQuantity := 0.0;
   END_IF;
END_REGION
END_FUNCTION_BLOCK
